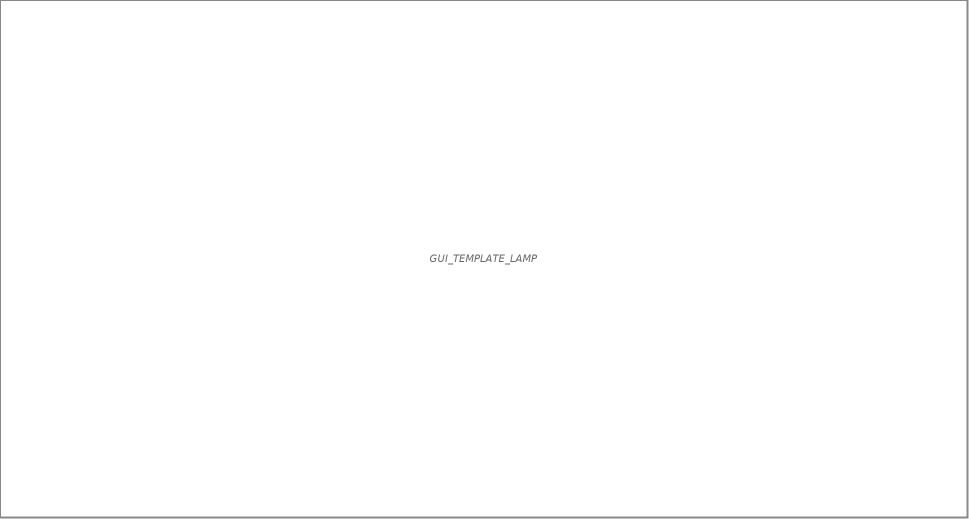
VISUALIZATION GUI_Lamp002  // 969x519
    Frame (0,0 967x517)
        shows GUI_TEMPLATE_LAMP(m_Instance := MAIN.Lamp002)
END_VISUALIZATION

(* stored: Version 1.1.0.1, ProductVersion 3.1.4024.3
   Visu GUI_Lamp002: Id {5c59290c-ae13-438f-9802-7936bb004608} *)
